FUNCTION_BLOCK AOI_DO
VAR_INPUT
	ON: BOOL;
	OFF: BOOL;
	NAME: STRING := 'Not use';
	VALUE: BOOL;
END_VAR
VAR_OUTPUT
	LINK: BOOL;
	R_TRIG: BOOL;
	F_TRIG: BOOL;
END_VAR
VAR
	rtON: R_TRIG;
	rtOFF: R_TRIG;
	rtValue: R_TRIG;
	ftValue: F_TRIG;
END_VAR

LINK:=  (ON OR  VALUE)   AND NOT OFF; 

rtValue(CLK:=VALUE);
ftValue(CLK:=VALUE);
R_TRIG:=rtValue.Q;
F_TRIG:=ftValue.Q;
rtON(CLK:=ON);
(*
IF rtON.Q THEN
	OFF:=FALSE;
	On:=TRUE;
END_IF
rtOFF(CLK:=OFF);
IF rtOFF.Q THEN
	ON:=FALSE;
	OFF:=TRUE;
END_IF
*)
IF on AND off THEN
	ON:=FALSE;
	OFF:=FALSE;	
END_IF

END_FUNCTION_BLOCK

(* stored: Version 1.1.0.1, ProductVersion 3.1.4024.6
   POU AOI_DO: Id {2a2adbd1-5365-40d2-9a23-ffd34a0a8e34}, SpecialFunc None *)
